// TIA Portal V17 export
// export: Created 2026-04-13T11:12:52.7396401Z, ExportSetting WithDefaults, DisplayName Totally Integrated Automation Portal, DisplayVersion V17 Update 4, DisplayName TIA Portal Openness, DisplayVersion V17 Update 4, DisplayName TIA Portal Version Control Interface, DisplayVersion V17, DisplayName SINAMICS Startdrive Advanced, DisplayVersion V17, DisplayName SINAMICS Startdrive G130, G150, S120, S150, SINAMICS MV, S210, DisplayVersion V17, DisplayName SINAMICS Startdrive G110M, G120, G120C, G120D, G120P, G115D, DisplayVersion V17, DisplayName STEP 7 Professional, DisplayVersion V17 Update 4, DisplayName STEP 7 Safety, DisplayVersion V17, DisplayName WinCC Professional, DisplayVersion V17 Update 4
TagTable "OUTCIPRJ"
  OUTCIPRJ_1设定时间 : Real  (PLC tag OUTCIPRJ.1设定时间, HMI_连接_1, 1 s)
  OUTCIPRJ_2设定时间 : Real  (PLC tag OUTCIPRJ.2设定时间, HMI_连接_1, 1 s)
  OUTCIPRJ_3设定时间 : Real  (PLC tag OUTCIPRJ.3设定时间, HMI_连接_1, 1 s)
  OUTCIPRJ_4设定时间 : Real  (PLC tag OUTCIPRJ.4设定时间, HMI_连接_1, 1 s)
  OUTCIPRJ_5设定时间 : Real  (PLC tag OUTCIPRJ.5设定时间, HMI_连接_1, 1 s)
  OUTCIPRJ_6设定时间 : Real  (PLC tag OUTCIPRJ.6设定时间, HMI_连接_1, 1 s)
  OUTCIPRJ_7设定时间 : Real  (PLC tag OUTCIPRJ.7设定时间, HMI_连接_1, 1 s)
  OUTCIPRJ_8设定时间 : Real  (PLC tag OUTCIPRJ.8设定时间, HMI_连接_1, 1 s)
  OUTCIPRJ_9设定时间 : Real  (PLC tag OUTCIPRJ.9设定时间, HMI_连接_1, 1 s)
  OUTCIPRJ_10设定时间 : Real  (PLC tag OUTCIPRJ.10设定时间, HMI_连接_1, 1 s)
  OUTCIPRJ_11设定时间 : Real  (PLC tag OUTCIPRJ.11设定时间, HMI_连接_1, 1 s)
  OUTCIPRJ_12设定时间 : Real  (PLC tag OUTCIPRJ.12设定时间, HMI_连接_1, 1 s)
  OUTCIPRJ_13设定时间 : Real  (PLC tag OUTCIPRJ.13设定时间, HMI_连接_1, 1 s)
  OUTCIPRJ_14设定时间 : Real  (PLC tag OUTCIPRJ.14设定时间, HMI_连接_1, 1 s)
  OUTCIPRJ_15设定时间 : Real  (PLC tag OUTCIPRJ.15设定时间, HMI_连接_1, 1 s)
  OUTCIPRJ_16设定时间 : Real  (PLC tag OUTCIPRJ.16设定时间, HMI_连接_1, 1 s)
  OUTCIPRJ_1计时 : Real  (PLC tag OUTCIPRJ.1计时, HMI_连接_1, 1 s)
  OUTCIPRJ_2计时 : Real  (PLC tag OUTCIPRJ.2计时, HMI_连接_1, 1 s)
  OUTCIPRJ_3计时 : Real  (PLC tag OUTCIPRJ.3计时, HMI_连接_1, 1 s)
  OUTCIPRJ_4计时 : Real  (PLC tag OUTCIPRJ.4计时, HMI_连接_1, 1 s)
  OUTCIPRJ_5计时 : Real  (PLC tag OUTCIPRJ.5计时, HMI_连接_1, 1 s)
  OUTCIPRJ_6计时 : Real  (PLC tag OUTCIPRJ.6计时, HMI_连接_1, 1 s)
  OUTCIPRJ_7计时 : Real  (PLC tag OUTCIPRJ.7计时, HMI_连接_1, 1 s)
  OUTCIPRJ_8计时 : Real  (PLC tag OUTCIPRJ.8计时, HMI_连接_1, 1 s)
  OUTCIPRJ_9计时 : Real  (PLC tag OUTCIPRJ.9计时, HMI_连接_1, 1 s)
  OUTCIPRJ_10计时 : Real  (PLC tag OUTCIPRJ.10计时, HMI_连接_1, 1 s)
  OUTCIPRJ_11计时 : Real  (PLC tag OUTCIPRJ.11计时, HMI_连接_1, 1 s)
  OUTCIPRJ_12计时 : Real  (PLC tag OUTCIPRJ.12计时, HMI_连接_1, 1 s)
  OUTCIPRJ_13计时 : Real  (PLC tag OUTCIPRJ.13计时, HMI_连接_1, 1 s)
  OUTCIPRJ_14计时 : Real  (PLC tag OUTCIPRJ.14计时, HMI_连接_1, 1 s)
  OUTCIPRJ_15计时 : Real  (PLC tag OUTCIPRJ.15计时, HMI_连接_1, 1 s)
  OUTCIPRJ_16计时 : Real  (PLC tag OUTCIPRJ.16计时, HMI_连接_1, 1 s)
